{attribute 'qualified_only'}
{attribute 'strict'}
TYPE State :
(
	CheckEnable := 0,
	Initialize := 5,
	WaitForButton := 10,
	StartMaster := 20,
	Synchronization := 30,
	FinishAndStopMotors := 40,
	GearOut := 50,
	ErrorState := 999
	
);
END_TYPE

(* stored: Version 1.1.0.1, ProductVersion 3.1.4024.12
   DUT State: Id {4ca2b2e0-0669-4687-bc4a-0ca73d9508f9} *)
